// Mitsubishi GX Works2 project: Jog   PLC: Q02/Q02H

// task Task_01 (event TRUE, interval 0, priority 31): POU_01

PROGRAM POU_01
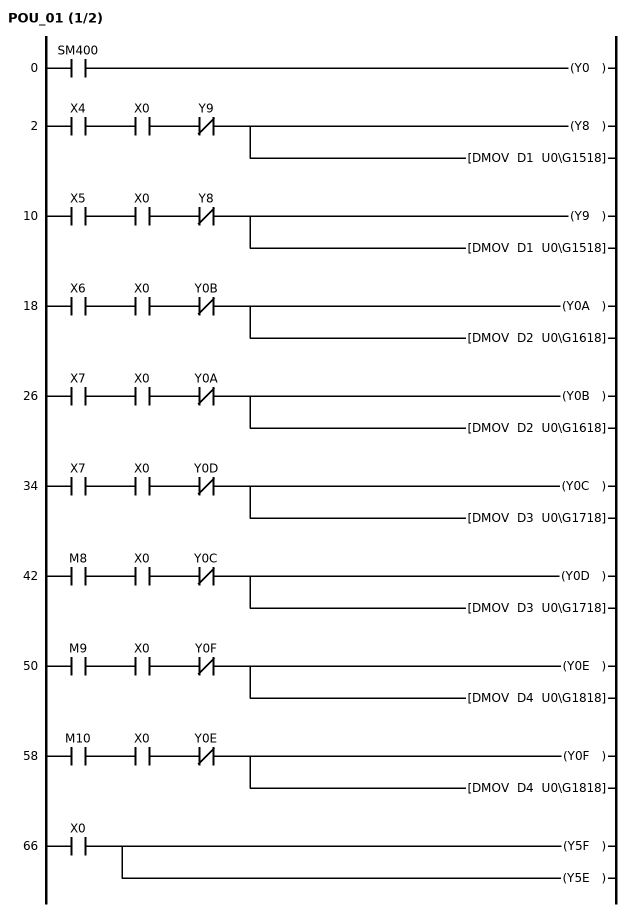
0     LD      SM400
      OUT     Y0
2     LD      X4
      AND     X0
      ANI     Y9
      OUT     Y8
      DMOV    D1 U0\G1518
10    LD      X5
      AND     X0
      ANI     Y8
      OUT     Y9
      DMOV    D1 U0\G1518
18    LD      X6
      AND     X0
      ANI     Y0B
      OUT     Y0A
      DMOV    D2 U0\G1618
26    LD      X7
      AND     X0
      ANI     Y0A
      OUT     Y0B
      DMOV    D2 U0\G1618
34    LD      X7
      AND     X0
      ANI     Y0D
      OUT     Y0C
      DMOV    D3 U0\G1718
42    LD      M8
      AND     X0
      ANI     Y0C
      OUT     Y0D
      DMOV    D3 U0\G1718
50    LD      M9
      AND     X0
      ANI     Y0F
      OUT     Y0E
      DMOV    D4 U0\G1818
58    LD      M10
      AND     X0
      ANI     Y0E
      OUT     Y0F
      DMOV    D4 U0\G1818
66    LD      X0
      OUT     Y5F
      OUT     Y5E
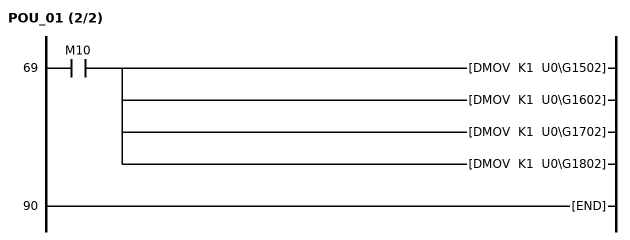
69    LD      M10
      DMOV    K1 U0\G1502
      DMOV    K1 U0\G1602
      DMOV    K1 U0\G1702
      DMOV    K1 U0\G1802
90    END
END_PROGRAM
